TYPE MotorOutputVariables :
STRUCT
	coil : BOOL;

END_STRUCT
END_TYPE

(* stored: Version 1.1.0.1, ProductVersion 3.1.4024.12
   DUT MotorOutputVariables: Id {5a034cf0-ad6a-4eed-872f-78c51913ee6d} *)
